(* IEC 61131-3 sources: GOPLC-Showcase/examples/st, 14 files *)

(* ---- alarm_handler.st ---- *)
(* ============================================================================
   Alarm Management System
   ============================================================================
   Industrial alarm handling with:
   - Multiple alarm priorities (Critical, High, Medium, Low)
   - Alarm acknowledgment and reset
   - Alarm history logging
   - Alarm shelving with timeout
   - Alarm suppression during mode changes
   ============================================================================ *)

VAR_GLOBAL
    (* Alarm inputs *)
    AI_HighTemp : BOOL := FALSE;
    AI_LowTemp : BOOL := FALSE;
    AI_HighPressure : BOOL := FALSE;
    AI_LowPressure : BOOL := FALSE;
    AI_LowLevel : BOOL := FALSE;
    AI_HighLevel : BOOL := FALSE;
    AI_MotorFault : BOOL := FALSE;
    AI_CommFault : BOOL := FALSE;

    (* Alarm outputs *)
    AO_AlarmActive : BOOL := FALSE;
    AO_AlarmCount : INT := 0;
    AO_HighestPriority : INT := 0;
    AO_Horn : BOOL := FALSE;
    AO_Beacon : BOOL := FALSE;

    (* Operator actions *)
    CMD_Acknowledge : BOOL := FALSE;
    CMD_SilenceHorn : BOOL := FALSE;
    CMD_Reset : BOOL := FALSE;
END_VAR

PROGRAM AlarmHandler
VAR
    (* Alarm state array: 0=Normal, 1=Active, 2=Acknowledged, 3=Shelved *)
    alarmState : ARRAY[0..7] OF INT;

    (* Alarm priorities: 1=Critical, 2=High, 3=Medium, 4=Low *)
    alarmPriority : ARRAY[0..7] OF INT := [1, 3, 2, 3, 3, 2, 1, 2];

    (* Alarm names for logging *)
    alarmNames : ARRAY[0..7] OF STRING := [
        'High Temperature',
        'Low Temperature',
        'High Pressure',
        'Low Pressure',
        'Low Level',
        'High Level',
        'Motor Fault',
        'Comm Fault'
    ];

    (* Alarm conditions *)
    alarmConditions : ARRAY[0..7] OF BOOL;

    (* Timing *)
    hornTimer : INT := 0;
    HORN_TIMEOUT : INT := 300;  (* Auto-silence after 30 seconds at 100ms scan *)

    (* Counters *)
    i : INT;
    activeCount : INT;
    highestPrio : INT;

    (* Edge detection for acknowledge *)
    ackPrev : BOOL := FALSE;
    resetPrev : BOOL := FALSE;
END_VAR

(* === Map Inputs to Alarm Conditions === *)
alarmConditions[0] := AI_HighTemp;
alarmConditions[1] := AI_LowTemp;
alarmConditions[2] := AI_HighPressure;
alarmConditions[3] := AI_LowPressure;
alarmConditions[4] := AI_LowLevel;
alarmConditions[5] := AI_HighLevel;
alarmConditions[6] := AI_MotorFault;
alarmConditions[7] := AI_CommFault;

(* === Process Each Alarm === *)
activeCount := 0;
highestPrio := 99;

FOR i := 0 TO 7 DO
    CASE alarmState[i] OF
        0: (* Normal *)
            IF alarmConditions[i] THEN
                alarmState[i] := 1;  (* Transition to Active *)
                (* Log alarm activation *)
                DEBUG_INFO(CONCAT('ALARM ACTIVE: ', alarmNames[i]));
            END_IF;

        1: (* Active - Unacknowledged *)
            IF NOT alarmConditions[i] THEN
                alarmState[i] := 0;  (* Return to normal *)
                DEBUG_INFO(CONCAT('ALARM CLEARED: ', alarmNames[i]));
            ELSIF CMD_Acknowledge AND NOT ackPrev THEN
                alarmState[i] := 2;  (* Acknowledged *)
                DEBUG_INFO(CONCAT('ALARM ACKED: ', alarmNames[i]));
            END_IF;

        2: (* Acknowledged *)
            IF NOT alarmConditions[i] THEN
                alarmState[i] := 0;  (* Return to normal *)
                DEBUG_INFO(CONCAT('ALARM CLEARED: ', alarmNames[i]));
            END_IF;

        3: (* Shelved *)
            (* Shelved alarms handled separately *)
            ;
    END_CASE;

    (* Count active alarms and find highest priority *)
    IF alarmState[i] = 1 OR alarmState[i] = 2 THEN
        activeCount := activeCount + 1;
        IF alarmPriority[i] < highestPrio THEN
            highestPrio := alarmPriority[i];
        END_IF;
    END_IF;
END_FOR;

(* === Update Outputs === *)
AO_AlarmCount := activeCount;
AO_AlarmActive := activeCount > 0;

IF activeCount > 0 THEN
    AO_HighestPriority := highestPrio;
ELSE
    AO_HighestPriority := 0;
END_IF;

(* === Horn Control === *)
(* Horn sounds for unacknowledged alarms *)
IF AO_AlarmActive THEN
    (* Check for any unacknowledged alarm *)
    FOR i := 0 TO 7 DO
        IF alarmState[i] = 1 THEN
            AO_Horn := TRUE;
            EXIT;
        END_IF;
    END_FOR;

    (* Auto-silence timeout *)
    IF AO_Horn THEN
        hornTimer := hornTimer + 1;
        IF hornTimer > HORN_TIMEOUT OR CMD_SilenceHorn THEN
            AO_Horn := FALSE;
        END_IF;
    END_IF;
ELSE
    AO_Horn := FALSE;
    hornTimer := 0;
END_IF;

(* === Beacon Control === *)
(* Beacon on for Critical (1) or High (2) priority active alarms *)
AO_Beacon := AO_AlarmActive AND (AO_HighestPriority <= 2);

(* === Reset Command === *)
IF CMD_Reset AND NOT resetPrev THEN
    FOR i := 0 TO 7 DO
        IF NOT alarmConditions[i] THEN
            alarmState[i] := 0;
        END_IF;
    END_FOR;
    DEBUG_INFO('ALARM SYSTEM RESET');
END_IF;

(* === Edge Detection Update === *)
ackPrev := CMD_Acknowledge;
resetPrev := CMD_Reset;

(* === Map to I/O === *)
%QX1.0 := AO_AlarmActive;
%QX1.1 := AO_Horn;
%QX1.2 := AO_Beacon;
%QW10 := AO_AlarmCount;
%QW11 := AO_HighestPriority;

(* Read operator commands *)
CMD_Acknowledge := %IX1.0;
CMD_SilenceHorn := %IX1.1;
CMD_Reset := %IX1.2;

END_PROGRAM

(* ---- bacnet_client.st ---- *)
// BACnet/IP Client Example
// Connects to a BACnet server and reads standard object types
PROGRAM BACnet_Client
VAR
    state       : DINT := 0;
    connected   : BOOL := FALSE;
    temp_zone1  : REAL;
    temp_zone2  : REAL;
    fan_status  : BOOL;
    setpoint    : REAL;
    tick_val    : REAL;
    prev_tick   : REAL;
    tick_live   : BOOL;
    cycles      : DINT := 0;
END_VAR

CASE state OF
    0: (* INIT — create BACnet client *)
        IF BACNET_CLIENT_CREATE('bac1', '10.0.0.100', 999, 0, 47808) THEN
            BACNET_CLIENT_CONNECT('bac1');
            state := 1;
        END_IF;

    1: (* WAIT FOR CONNECTION *)
        IF BACNET_CLIENT_IS_CONNECTED('bac1') THEN
            state := 10;
        END_IF;

    10: (* RUNNING — read BACnet objects *)
        temp_zone1 := BACNET_READ_AI('bac1', 0);
        temp_zone2 := BACNET_READ_AI('bac1', 1);
        fan_status := BACNET_READ_BI('bac1', 0);
        setpoint   := BACNET_READ_AV('bac1', 0);
        tick_val   := BACNET_READ_AI('bac1', 2);

        tick_live  := tick_val <> prev_tick;
        prev_tick  := tick_val;
        cycles     := cycles + 1;

    ELSE
        state := 0;
END_CASE;
END_PROGRAM

(* ---- data_sync.st ---- *)
(* ============================================================================
   Multi-PLC Data Synchronization
   ============================================================================
   Demonstrates GOPLC's DataLayer for real-time variable sharing:
   - Publish local variables to other PLCs
   - Subscribe to variables from remote PLCs
   - Measure synchronization latency
   - Handle communication failures gracefully
   ============================================================================ *)

VAR_GLOBAL
    (* Local variables - published to other PLCs *)
    LOCAL_Counter : DINT := 0;
    LOCAL_Temperature : REAL := 0.0;
    LOCAL_Pressure : REAL := 0.0;
    LOCAL_Status : INT := 0;
    LOCAL_Alarm : BOOL := FALSE;

    (* Remote variables - received from PLC2 *)
    REMOTE_PLC2_Counter : DINT := 0;
    REMOTE_PLC2_Temperature : REAL := 0.0;
    REMOTE_PLC2_Status : INT := 0;

    (* Sync diagnostics *)
    SYNC_Latency_us : DINT := 0;
    SYNC_LastUpdate_ms : DINT := 0;
    SYNC_CommOK : BOOL := FALSE;
END_VAR

PROGRAM DataSync
VAR
    (* Simulation state *)
    simAngle : REAL := 0.0;
    scanCount : DINT := 0;

    (* Communication monitoring *)
    lastRemoteCounter : DINT := 0;
    commTimeout : INT := 0;
    COMM_TIMEOUT_LIMIT : INT := 100;  (* 100 scans without update = fault *)

    (* Calculated values *)
    avgTemperature : REAL := 0.0;
    tempDiff : REAL := 0.0;
END_VAR

(* === Increment Local Counter === *)
scanCount := scanCount + 1;
LOCAL_Counter := scanCount;

(* === Simulate Local Sensor Data === *)
simAngle := simAngle + 0.05;
IF simAngle > 6.28 THEN
    simAngle := 0.0;
END_IF;

(* Temperature: 20-30C with sine wave variation *)
LOCAL_Temperature := 25.0 + 5.0 * SIN(simAngle);

(* Pressure: 100-110 kPa with cosine variation *)
LOCAL_Pressure := 105.0 + 5.0 * COS(simAngle * 0.7);

(* Status: 0=OK, 1=Warning, 2=Alarm *)
IF LOCAL_Temperature > 28.0 THEN
    LOCAL_Status := 1;
    LOCAL_Alarm := FALSE;
ELSIF LOCAL_Temperature > 29.5 THEN
    LOCAL_Status := 2;
    LOCAL_Alarm := TRUE;
ELSE
    LOCAL_Status := 0;
    LOCAL_Alarm := FALSE;
END_IF;

(* === Read Remote Variables via DataLayer === *)
(* These are automatically populated by the DataLayer subscription *)
(* Check if we're receiving updates from PLC2 *)

IF REMOTE_PLC2_Counter <> lastRemoteCounter THEN
    (* Got new data from PLC2 *)
    lastRemoteCounter := REMOTE_PLC2_Counter;
    commTimeout := 0;
    SYNC_CommOK := TRUE;

    (* Measure sync latency *)
    SYNC_Latency_us := DL_LATENCY_US('plc2', 'LOCAL_Counter');
    SYNC_LastUpdate_ms := DINT_TO_INT(TICK_MS() MOD 100000);
ELSE
    (* No update this scan *)
    commTimeout := commTimeout + 1;
    IF commTimeout > COMM_TIMEOUT_LIMIT THEN
        SYNC_CommOK := FALSE;
    END_IF;
END_IF;

(* === Calculate Cross-PLC Metrics === *)
IF SYNC_CommOK THEN
    (* Average temperature across both PLCs *)
    avgTemperature := (LOCAL_Temperature + REMOTE_PLC2_Temperature) / 2.0;

    (* Temperature difference for load balancing *)
    tempDiff := ABS(LOCAL_Temperature - REMOTE_PLC2_Temperature);
END_IF;

(* === Map to Modbus Registers === *)
%QW0 := DINT_TO_INT(LOCAL_Counter MOD 32767);
%QW1 := REAL_TO_INT(LOCAL_Temperature * 10.0);
%QW2 := REAL_TO_INT(LOCAL_Pressure * 10.0);
%QW3 := LOCAL_Status;
%QW4 := DINT_TO_INT(REMOTE_PLC2_Counter MOD 32767);
%QW5 := REAL_TO_INT(REMOTE_PLC2_Temperature * 10.0);
%QW6 := DINT_TO_INT(SYNC_Latency_us MOD 32767);
%QX0.0 := SYNC_CommOK;
%QX0.1 := LOCAL_Alarm;

END_PROGRAM

(* ---- datalayer_ethercat.st ---- *)
// ctrlX Data Layer — EtherCAT I/O via Native IPC
// Reads digital inputs and toggles digital outputs on ctrlX CORE
PROGRAM DataLayer_EtherCat
VAR
    state       : DINT := 0;
    connected   : BOOL := FALSE;
    di1         : BOOL := FALSE;
    di2         : BOOL := FALSE;
    di3         : BOOL := FALSE;
    di4         : BOOL := FALSE;
    do1         : BOOL := FALSE;
    toggle      : BOOL := FALSE;
    toggle_tmr  : TON;
    write_ok    : BOOL := FALSE;
    stats       : STRING := '';
    tick        : DINT := 0;
END_VAR

CASE state OF
    0: (* INIT — create EtherCAT connection, native IPC mode *)
        IF CTRLX_EC_CREATE('ec1', '', '', '', 'XI110116', 'XI211116', 16, 16, 10, 'dl') THEN
            CTRLX_EC_START('ec1');
            state := 10;
        END_IF;

    10: (* RUNNING — read inputs, toggle outputs *)
        connected := CTRLX_EC_CONNECTED('ec1');
        IF NOT connected THEN
            state := 0;
        END_IF;

        di1 := CTRLX_EC_READ_DI('ec1', 1);
        di2 := CTRLX_EC_READ_DI('ec1', 2);
        di3 := CTRLX_EC_READ_DI('ec1', 3);
        di4 := CTRLX_EC_READ_DI('ec1', 4);

        // Toggle output every 100ms
        toggle_tmr(IN := NOT toggle_tmr.Q, PT := T#100ms);
        IF toggle_tmr.Q THEN
            toggle := NOT toggle;
        END_IF;

        write_ok := CTRLX_EC_WRITE_DO('ec1', 1, toggle);
        do1 := CTRLX_EC_READ_DO('ec1', 1);
        stats := CTRLX_EC_STATS('ec1');
        tick := tick + 1;

    ELSE
        state := 0;
END_CASE;
END_PROGRAM

(* ---- dnp3_master.st ---- *)
// DNP3 Master Example
// Connects to a utility outstation (RTU) and reads/writes points
PROGRAM DNP3_Master
VAR
    state       : DINT := 0;
    connected   : BOOL := FALSE;
    // Analog inputs — field measurements
    flow_rate   : REAL;
    pressure    : REAL;
    level       : REAL;
    // Binary inputs — equipment status
    pump_run    : BOOL;
    valve_open  : BOOL;
    alarm_hi    : BOOL;
    // Control outputs
    pump_cmd    : BOOL := FALSE;
    setpoint    : REAL := 50.0;
    write_ok    : BOOL;
    counter     : INT;
    cycles      : DINT := 0;
END_VAR

CASE state OF
    0: (* INIT — create DNP3 master, local addr 1, remote addr 10 *)
        IF DNP3_MASTER_CREATE('rtu1', '10.0.0.100', 20000, 1, 10) THEN
            state := 1;
        END_IF;

    1: (* CONNECT *)
        IF DNP3_MASTER_CONNECT('rtu1') THEN
            state := 10;
        END_IF;

    10: (* RUNNING — poll field data *)
        connected := DNP3_MASTER_IS_CONNECTED('rtu1');
        IF NOT connected THEN
            state := 1;
        END_IF;

        // Read analog inputs (field instruments)
        flow_rate := DNP3_MASTER_READ_AI('rtu1', 0);
        pressure  := DNP3_MASTER_READ_AI('rtu1', 1);
        level     := DNP3_MASTER_READ_AI('rtu1', 2);

        // Read binary inputs (equipment status)
        pump_run   := DNP3_MASTER_READ_BI('rtu1', 0);
        valve_open := DNP3_MASTER_READ_BI('rtu1', 1);
        alarm_hi   := DNP3_MASTER_READ_BI('rtu1', 2);

        // Read counter
        counter := DNP3_MASTER_READ_COUNTER('rtu1', 0);

        // Write control outputs
        write_ok := DNP3_MASTER_WRITE_BO('rtu1', 0, pump_cmd);
        DNP3_MASTER_WRITE_AO('rtu1', 0, setpoint);

        cycles := cycles + 1;

    ELSE
        state := 0;
END_CASE;
END_PROGRAM

(* ---- enip_scanner.st ---- *)
// EtherNet/IP Scanner Example
// Connects to a ControlLogix PLC and reads/writes CIP tags
PROGRAM ENIP_Scanner
VAR
    state       : DINT := 0;
    int_val     : INT;
    real_val    : REAL;
    bool_val    : BOOL;
    dint_val    : DINT;
    prev_int    : INT;
    changing    : BOOL;
    cycles      : DINT := 0;
END_VAR

CASE state OF
    0: (* INIT — create scanner with tag list *)
        IF ENIP_SCANNER_CREATE('plc1', '10.0.0.100', 44818) THEN
            ENIP_SCANNER_ADD_INT_TAG('plc1', 'Speed_SP', 1);
            ENIP_SCANNER_ADD_REAL_TAG('plc1', 'Temperature', 1);
            ENIP_SCANNER_ADD_BOOL_TAG('plc1', 'RunStatus', 1);
            ENIP_SCANNER_ADD_DINT_TAG('plc1', 'TotalCount', 1);
            ENIP_SCANNER_CONNECT('plc1');
            state := 10;
        END_IF;

    10: (* RUNNING — read tags *)
        int_val  := ENIP_SCANNER_READ_INT('plc1', 'Speed_SP', 0);
        real_val := ENIP_SCANNER_READ_REAL('plc1', 'Temperature', 0);
        bool_val := ENIP_SCANNER_READ_BOOL('plc1', 'RunStatus', 0);
        dint_val := ENIP_SCANNER_READ_DINT('plc1', 'TotalCount', 0);

        changing := int_val <> prev_int;
        prev_int := int_val;
        cycles   := cycles + 1;

    ELSE
        state := 0;
END_CASE;
END_PROGRAM

(* ---- esp32_io.st ---- *)
(* ============================================================================
   ESP32 Remote I/O Controller
   ============================================================================
   Control an ESP32-S3 running as a Modbus TCP I/O module:
   - 8 Digital Inputs
   - 8 Digital Outputs
   - 3 Analog Inputs (12-bit ADC)
   - 2 PWM Outputs
   - RGB NeoPixel LED
   ============================================================================ *)

PROGRAM ESP32_IO
VAR
    (* Digital Inputs from ESP32 *)
    DI0 AT %IX0.0 : BOOL;
    DI1 AT %IX0.1 : BOOL;
    DI2 AT %IX0.2 : BOOL;
    DI3 AT %IX0.3 : BOOL;
    DI4 AT %IX0.4 : BOOL;
    DI5 AT %IX0.5 : BOOL;
    DI6 AT %IX0.6 : BOOL;
    DI7 AT %IX0.7 : BOOL;

    (* Digital Outputs to ESP32 *)
    DO0 AT %QX0.0 : BOOL;
    DO1 AT %QX0.1 : BOOL;
    DO2 AT %QX0.2 : BOOL;
    DO3 AT %QX0.3 : BOOL;
    DO4 AT %QX0.4 : BOOL;
    DO5 AT %QX0.5 : BOOL;
    DO6 AT %QX0.6 : BOOL;
    DO7 AT %QX0.7 : BOOL;

    (* ADC Inputs (12-bit, 0-4095) *)
    ADC0 AT %IW0 : INT;
    ADC1 AT %IW1 : INT;
    ADC2 AT %IW2 : INT;

    (* PWM Outputs (0-1023) *)
    PWM0 AT %QW0 : INT;
    PWM1 AT %QW1 : INT;

    (* RGB LED (0-255 each) *)
    LED_R AT %QW10 : INT;
    LED_G AT %QW11 : INT;
    LED_B AT %QW12 : INT;

    (* Calculated values *)
    ADC0_Volts : REAL;
    ADC1_Volts : REAL;
    ADC2_Volts : REAL;

    (* Demo state *)
    Heartbeat : BOOL := FALSE;
    Counter : INT := 0;
    ColorPhase : INT := 0;
END_VAR

(* === Heartbeat Output === *)
Heartbeat := NOT Heartbeat;
DO0 := Heartbeat;

(* === Convert ADC to Voltage === *)
(* ESP32 ADC: 3.3V reference, 12-bit resolution *)
ADC0_Volts := INT_TO_REAL(ADC0) * 3.3 / 4095.0;
ADC1_Volts := INT_TO_REAL(ADC1) * 3.3 / 4095.0;
ADC2_Volts := INT_TO_REAL(ADC2) * 3.3 / 4095.0;

(* === PWM Based on ADC === *)
(* Map ADC0 (0-4095) to PWM0 (0-1023) *)
PWM0 := ADC0 / 4;

(* Map ADC1 to PWM1 with deadband *)
IF ADC1 > 200 THEN
    PWM1 := (ADC1 - 200) / 4;
ELSE
    PWM1 := 0;
END_IF;

(* === RGB LED Color Cycle === *)
Counter := Counter + 1;
IF Counter > 50 THEN
    Counter := 0;
    ColorPhase := ColorPhase + 1;
    IF ColorPhase > 5 THEN
        ColorPhase := 0;
    END_IF;
END_IF;

CASE ColorPhase OF
    0: (* Red *)
        LED_R := 50; LED_G := 0; LED_B := 0;
    1: (* Yellow *)
        LED_R := 50; LED_G := 30; LED_B := 0;
    2: (* Green *)
        LED_R := 0; LED_G := 50; LED_B := 0;
    3: (* Cyan *)
        LED_R := 0; LED_G := 50; LED_B := 50;
    4: (* Blue *)
        LED_R := 0; LED_G := 0; LED_B := 50;
    5: (* Magenta *)
        LED_R := 50; LED_G := 0; LED_B := 50;
END_CASE;

(* Override color based on input *)
IF DI1 THEN
    (* Input 1 = Force Red (alarm) *)
    LED_R := 255; LED_G := 0; LED_B := 0;
ELSIF DI2 THEN
    (* Input 2 = Force Green (OK) *)
    LED_R := 0; LED_G := 255; LED_B := 0;
END_IF;

(* === Digital Output Loopback === *)
DO1 := DI0;
DO2 := DI1;
DO3 := DI2;

END_PROGRAM

(* ---- fins_client.st ---- *)
// Omron FINS Client Example
// Reads/writes DM (Data Memory) words on an Omron PLC
PROGRAM FINS_Client
VAR
    state       : DINT := 0;
    dm_data     : ARRAY[0..10] OF INT;
    prev_tick   : INT;
    tick_live   : BOOL;
    write_ok    : BOOL;
    readback    : ARRAY[0..1] OF INT;
    write_pass  : BOOL;
    cycles      : DINT := 0;
END_VAR

CASE state OF
    0: (* INIT — connect to Omron PLC *)
        IF FINS_CLIENT_CREATE('omron1', '10.0.0.100', 9600) THEN
            FINS_CLIENT_CONNECT('omron1');
            state := 10;
        END_IF;

    10: (* RUNNING — bulk read DM, write-back test *)
        dm_data := FINS_CLIENT_READ_DM('omron1', 0, 11);

        tick_live := dm_data[10] <> prev_tick;
        prev_tick := dm_data[10];

        // Write a value and read it back to verify
        write_ok  := FINS_CLIENT_WRITE_DM_WORD('omron1', 20, 8888);
        readback  := FINS_CLIENT_READ_DM('omron1', 20, 2);
        write_pass := readback[0] = 8888;

        cycles := cycles + 1;

    ELSE
        state := 0;
END_CASE;
END_PROGRAM

(* ---- iec104_client.st ---- *)
// IEC 60870-5-104 Client Example
// Connects to a utility SCADA outstation and reads telemetry
PROGRAM IEC104_Client
VAR
    state       : DINT := 0;
    sp1         : BOOL;
    sp2         : BOOL;
    float_val   : REAL;
    scaled_val  : INT;
    counter_val : INT;
    tick_val    : INT;
    prev_tick   : INT;
    tick_live   : BOOL;
    cycles      : DINT := 0;
END_VAR

CASE state OF
    0: (* INIT — connect to IEC 104 outstation *)
        IF IEC104_CLIENT_CREATE('rtu1', '10.0.0.100', 2404) THEN
            IEC104_CLIENT_CONNECT('rtu1');
            state := 10;
        END_IF;

    10: (* RUNNING — read telemetry *)
        sp1        := IEC104_CLIENT_READ_SP('rtu1', 1);
        sp2        := IEC104_CLIENT_READ_SP('rtu1', 2);
        float_val  := IEC104_CLIENT_READ_FLOAT('rtu1', 10);
        scaled_val := IEC104_CLIENT_READ_SCALED('rtu1', 20);
        counter_val := IEC104_CLIENT_READ_COUNTER('rtu1', 30);
        tick_val   := IEC104_CLIENT_READ_COUNTER('rtu1', 31);

        tick_live  := tick_val <> prev_tick;
        prev_tick  := tick_val;
        cycles     := cycles + 1;

    ELSE
        state := 0;
END_CASE;
END_PROGRAM

(* ---- modbus_client.st ---- *)
// Modbus TCP Client Example
// Reads holding registers, input registers, and coils from a Modbus server
PROGRAM Modbus_Client
VAR
    state       : DINT := 0;
    hr_data     : ARRAY[0..10] OF INT;
    ir_data     : ARRAY[0..1] OF INT;
    coils       : ARRAY[0..2] OF BOOL;
    prev_tick   : INT;
    tick_live   : BOOL;
    write_ok    : BOOL;
    readback    : ARRAY[0..1] OF INT;
    write_pass  : BOOL;
    cycles      : DINT := 0;
END_VAR

CASE state OF
    0: (* INIT — connect to Modbus server *)
        IF MB_CLIENT_CREATE('mb1', '10.0.0.100', 502) THEN
            MB_CLIENT_CONNECT('mb1');
            state := 10;
        END_IF;

    10: (* RUNNING — read registers and coils *)
        hr_data := MB_READ_HOLDING('mb1', 0, 11);
        ir_data := MB_READ_INPUT('mb1', 0, 2);
        coils   := MB_READ_COILS('mb1', 0, 3);

        tick_live := hr_data[10] <> prev_tick;
        prev_tick := hr_data[10];

        // Write-back test
        write_ok  := MB_WRITE_REGISTER('mb1', 20, 7777);
        readback  := MB_READ_HOLDING('mb1', 20, 2);
        write_pass := readback[0] = 7777;

        cycles := cycles + 1;

    ELSE
        state := 0;
END_CASE;
END_PROGRAM

(* ---- modbus_gateway.st ---- *)
(* ============================================================================
   Modbus Gateway - Bridge Between Modbus Devices
   ============================================================================
   This program demonstrates GOPLC's protocol bridging capabilities:
   - Read from remote Modbus TCP devices
   - Aggregate data into local registers
   - Expose via built-in Modbus server
   ============================================================================ *)

VAR_GLOBAL
    (* Gateway status *)
    GW_DevicesOnline : INT := 0;
    GW_TotalReads : DINT := 0;
    GW_TotalErrors : DINT := 0;
    GW_LastError : STRING := '';

    (* Aggregated sensor data *)
    Sensor_Temp_Zone1 : REAL := 0.0;
    Sensor_Temp_Zone2 : REAL := 0.0;
    Sensor_Temp_Zone3 : REAL := 0.0;
    Sensor_Humidity : REAL := 0.0;
    Sensor_Pressure : REAL := 0.0;

    (* Control outputs *)
    Control_Setpoint : REAL := 22.0;
    Control_Enable : BOOL := TRUE;
END_VAR

PROGRAM ModbusGateway
VAR
    (* Modbus client handles *)
    mbClient1 : DINT := 0;
    mbClient2 : DINT := 0;
    mbClient3 : DINT := 0;

    (* Polling state *)
    pollCycle : INT := 0;
    initialized : BOOL := FALSE;

    (* Read buffers *)
    rawTemp1 : INT;
    rawTemp2 : INT;
    rawTemp3 : INT;
    rawHumidity : INT;
    rawPressure : INT;

    (* Conversion constants *)
    TEMP_SCALE : REAL := 0.1;    (* Raw value * 0.1 = degrees C *)
    HUM_SCALE : REAL := 0.1;     (* Raw value * 0.1 = %RH *)
    PRESS_SCALE : REAL := 0.01;  (* Raw value * 0.01 = kPa *)
END_VAR

(* === Initialize Modbus Clients === *)
IF NOT initialized THEN
    (* Create client connections to remote devices *)
    mbClient1 := MB_CLIENT_CREATE('device1', '192.168.1.10', 502, 1);
    mbClient2 := MB_CLIENT_CREATE('device2', '192.168.1.11', 502, 1);
    mbClient3 := MB_CLIENT_CREATE('device3', '192.168.1.12', 502, 1);

    IF mbClient1 > 0 AND mbClient2 > 0 AND mbClient3 > 0 THEN
        initialized := TRUE;
        GW_DevicesOnline := 3;
    END_IF;
END_IF;

(* === Poll Devices in Round-Robin === *)
IF initialized THEN
    pollCycle := pollCycle + 1;
    IF pollCycle > 2 THEN
        pollCycle := 0;
    END_IF;

    CASE pollCycle OF
        0: (* Read Zone 1 Temperature from Device 1 *)
            IF MB_READ_HOLDING_REGISTERS(mbClient1, 0, 1, rawTemp1) THEN
                Sensor_Temp_Zone1 := INT_TO_REAL(rawTemp1) * TEMP_SCALE;
                GW_TotalReads := GW_TotalReads + 1;
            ELSE
                GW_TotalErrors := GW_TotalErrors + 1;
                GW_LastError := 'Device1 read failed';
            END_IF;

        1: (* Read Zone 2 & 3 from Device 2 *)
            IF MB_READ_HOLDING_REGISTERS(mbClient2, 0, 2, rawTemp2) THEN
                Sensor_Temp_Zone2 := INT_TO_REAL(rawTemp2) * TEMP_SCALE;
                Sensor_Temp_Zone3 := INT_TO_REAL(rawTemp3) * TEMP_SCALE;
                GW_TotalReads := GW_TotalReads + 1;
            ELSE
                GW_TotalErrors := GW_TotalErrors + 1;
                GW_LastError := 'Device2 read failed';
            END_IF;

        2: (* Read Humidity & Pressure from Device 3 *)
            IF MB_READ_HOLDING_REGISTERS(mbClient3, 0, 2, rawHumidity) THEN
                Sensor_Humidity := INT_TO_REAL(rawHumidity) * HUM_SCALE;
                Sensor_Pressure := INT_TO_REAL(rawPressure) * PRESS_SCALE;
                GW_TotalReads := GW_TotalReads + 1;
            ELSE
                GW_TotalErrors := GW_TotalErrors + 1;
                GW_LastError := 'Device3 read failed';
            END_IF;
    END_CASE;
END_IF;

(* === Map to Modbus Server Registers === *)
(* These are accessible via the built-in Modbus server *)
%QW0 := REAL_TO_INT(Sensor_Temp_Zone1 / TEMP_SCALE);
%QW1 := REAL_TO_INT(Sensor_Temp_Zone2 / TEMP_SCALE);
%QW2 := REAL_TO_INT(Sensor_Temp_Zone3 / TEMP_SCALE);
%QW3 := REAL_TO_INT(Sensor_Humidity / HUM_SCALE);
%QW4 := REAL_TO_INT(Sensor_Pressure / PRESS_SCALE);
%QW5 := REAL_TO_INT(Control_Setpoint / TEMP_SCALE);
%QW6 := GW_DevicesOnline;
%QW7 := DINT_TO_INT(GW_TotalReads MOD 32767);
%QW8 := DINT_TO_INT(GW_TotalErrors MOD 32767);

(* Read setpoint from external SCADA *)
Control_Setpoint := INT_TO_REAL(%IW0) * TEMP_SCALE;
Control_Enable := %IX0.0;

END_PROGRAM

(* ---- mqtt_publish.st ---- *)
// MQTT Publish/Subscribe Example
// Publishes telemetry and subscribes to command topics
PROGRAM MQTT_PubSub
VAR
    state        : DINT := 0;
    connected    : BOOL := FALSE;
    // Telemetry to publish
    temperature  : REAL := 22.5;
    humidity     : REAL := 45.0;
    pressure     : REAL := 1013.25;
    pub_ok       : BOOL;
    // Subscribed commands
    cmd_setpoint : REAL;
    cmd_enable   : BOOL;
    has_cmd      : BOOL;
    pub_tick     : DINT := 0;
    cycles       : DINT := 0;
END_VAR

CASE state OF
    0: (* INIT — connect to MQTT broker *)
        IF MQTT_CLIENT_CREATE('broker1', 'tcp://10.0.0.100:1883', 'goplc-plc01') THEN
            state := 1;
        END_IF;

    1: (* CONNECT and subscribe *)
        IF MQTT_CLIENT_CONNECT('broker1') THEN
            MQTT_SUBSCRIBE('broker1', 'plant/plc01/cmd/#');
            state := 10;
        END_IF;

    10: (* RUNNING — publish telemetry, check commands *)
        connected := MQTT_CLIENT_IS_CONNECTED('broker1');
        IF NOT connected THEN
            state := 1;
        END_IF;

        // Publish telemetry every 10 scans
        pub_tick := pub_tick + 1;
        IF pub_tick >= 10 THEN
            pub_tick := 0;
            MQTT_PUBLISH('broker1', 'plant/plc01/temperature', temperature);
            MQTT_PUBLISH('broker1', 'plant/plc01/humidity', humidity);
            pub_ok := MQTT_PUBLISH('broker1', 'plant/plc01/pressure', pressure);
        END_IF;

        // Check for incoming commands
        has_cmd := MQTT_HAS_MESSAGE('broker1', 'plant/plc01/cmd/setpoint');
        IF has_cmd THEN
            cmd_setpoint := MQTT_GET_MESSAGE_REAL('broker1', 'plant/plc01/cmd/setpoint');
        END_IF;

        cmd_enable := MQTT_GET_MESSAGE_BOOL('broker1', 'plant/plc01/cmd/enable');
        cycles := cycles + 1;

    ELSE
        state := 0;
END_CASE;
END_PROGRAM

(* ---- opcua_client.st ---- *)
// OPC UA Client Example
// Connects to an OPC UA server and reads/writes nodes
PROGRAM OPCUA_Client
VAR
    state       : DINT := 0;
    connected   : BOOL := FALSE;
    // Read values
    temperature : REAL;
    speed_sp    : INT;
    run_status  : BOOL;
    product_id  : STRING;
    // Write values
    new_setpoint : REAL := 75.0;
    write_ok    : BOOL;
    cycles      : DINT := 0;
END_VAR

CASE state OF
    0: (* INIT — create OPC UA client *)
        IF OPCUA_CLIENT_CREATE('srv1', 'opc.tcp://10.0.0.100:4840') THEN
            state := 1;
        END_IF;

    1: (* CONNECT *)
        IF OPCUA_CLIENT_CONNECT('srv1') THEN
            state := 10;
        END_IF;

    10: (* RUNNING — read and write nodes *)
        connected := OPCUA_CLIENT_IS_CONNECTED('srv1');
        IF NOT connected THEN
            state := 1;
        END_IF;

        // Read process values by Node ID
        temperature := OPCUA_CLIENT_READ_REAL('srv1', 'ns=2;s=Temperature');
        speed_sp    := OPCUA_CLIENT_READ_INT('srv1', 'ns=2;s=SpeedSetpoint');
        run_status  := OPCUA_CLIENT_READ_BOOL('srv1', 'ns=2;s=Running');
        product_id  := OPCUA_CLIENT_READ_STRING('srv1', 'ns=2;s=ProductID');

        // Write a setpoint
        write_ok := OPCUA_CLIENT_WRITE_REAL('srv1', 'ns=2;s=TempSetpoint', new_setpoint);

        cycles := cycles + 1;

    ELSE
        state := 0;
END_CASE;
END_PROGRAM

(* ---- pid_control.st ---- *)
(* ============================================================================
   PID Controller with Anti-Windup
   ============================================================================
   Industrial PID control with:
   - Proportional, Integral, Derivative terms
   - Anti-windup using back-calculation
   - Output clamping with configurable limits
   - Bumpless transfer on setpoint changes
   - Manual/Auto mode switching
   ============================================================================ *)

VAR_GLOBAL
    (* Process variables *)
    PV : REAL := 0.0;              (* Process Value - measured *)
    SP : REAL := 50.0;             (* Setpoint *)
    CV : REAL := 0.0;              (* Control Variable - output *)

    (* Tuning parameters *)
    Kp : REAL := 2.0;              (* Proportional gain *)
    Ki : REAL := 0.5;              (* Integral gain *)
    Kd : REAL := 0.1;              (* Derivative gain *)

    (* Limits *)
    CV_Max : REAL := 100.0;
    CV_Min : REAL := 0.0;

    (* Mode *)
    AutoMode : BOOL := TRUE;
    ManualCV : REAL := 0.0;

    (* Status *)
    Error : REAL := 0.0;
    Saturated : BOOL := FALSE;
END_VAR

PROGRAM PIDControl
VAR
    (* Internal state *)
    integral : REAL := 0.0;
    prevError : REAL := 0.0;
    prevPV : REAL := 0.0;
    derivative : REAL := 0.0;

    (* Anti-windup *)
    cvUnclamped : REAL := 0.0;
    backCalc : REAL := 0.0;
    Kb : REAL := 1.0;              (* Back-calculation gain *)

    (* Timing *)
    dt : REAL := 0.1;              (* Sample time in seconds *)

    (* Derivative filter *)
    derivFilt : REAL := 0.0;
    Tf : REAL := 0.05;             (* Filter time constant *)
END_VAR

(* === Calculate Error === *)
Error := SP - PV;

IF AutoMode THEN
    (* === Proportional Term === *)
    (* P = Kp * error *)

    (* === Integral Term with Anti-Windup === *)
    (* Only integrate if not saturated, or if integration would reduce saturation *)
    IF NOT Saturated OR (Error * integral < 0.0) THEN
        integral := integral + Ki * Error * dt;
        (* Back-calculation anti-windup *)
        integral := integral + Kb * backCalc * dt;
    END_IF;

    (* === Derivative Term (on PV to avoid derivative kick) === *)
    (* Use filtered derivative to reduce noise *)
    derivative := (PV - prevPV) / dt;
    derivFilt := derivFilt + (dt / Tf) * (derivative - derivFilt);

    (* === Calculate Unclamped Output === *)
    cvUnclamped := Kp * Error + integral - Kd * derivFilt;

    (* === Clamp Output === *)
    IF cvUnclamped > CV_Max THEN
        CV := CV_Max;
        Saturated := TRUE;
        backCalc := CV - cvUnclamped;
    ELSIF cvUnclamped < CV_Min THEN
        CV := CV_Min;
        Saturated := TRUE;
        backCalc := CV - cvUnclamped;
    ELSE
        CV := cvUnclamped;
        Saturated := FALSE;
        backCalc := 0.0;
    END_IF;

ELSE
    (* Manual mode - direct control *)
    CV := ManualCV;
    (* Track integral for bumpless transfer *)
    integral := CV - Kp * Error;
    Saturated := FALSE;
END_IF;

(* === Update Previous Values === *)
prevError := Error;
prevPV := PV;

(* === Map to I/O === *)
(* Output to analog output (0-100% = 0-10000) *)
%QW0 := REAL_TO_INT(CV * 100.0);

(* Read process value from analog input *)
PV := INT_TO_REAL(%IW0) / 100.0;

(* Read setpoint from HMI *)
SP := INT_TO_REAL(%IW1) / 10.0;

(* Mode from digital input *)
AutoMode := %IX0.0;

END_PROGRAM
